FUNCTION _TODO : BOOL
VAR_INPUT
END_VAR
VAR
END_VAR

// - ros2: specific check IF available
// - ros2: autoconfigure skill
// - opcua connecotr wrtie failed weil kein specific vorhanden war.
// - eyes skill: wird nie in state finalized gehen

END_FUNCTION

(* stored: Version 1.1.0.1, ProductVersion 3.1.4026.18
   POU _TODO: Id {066b45c6-4b88-4e09-8705-6da2621f10ea}, SpecialFunc None *)
